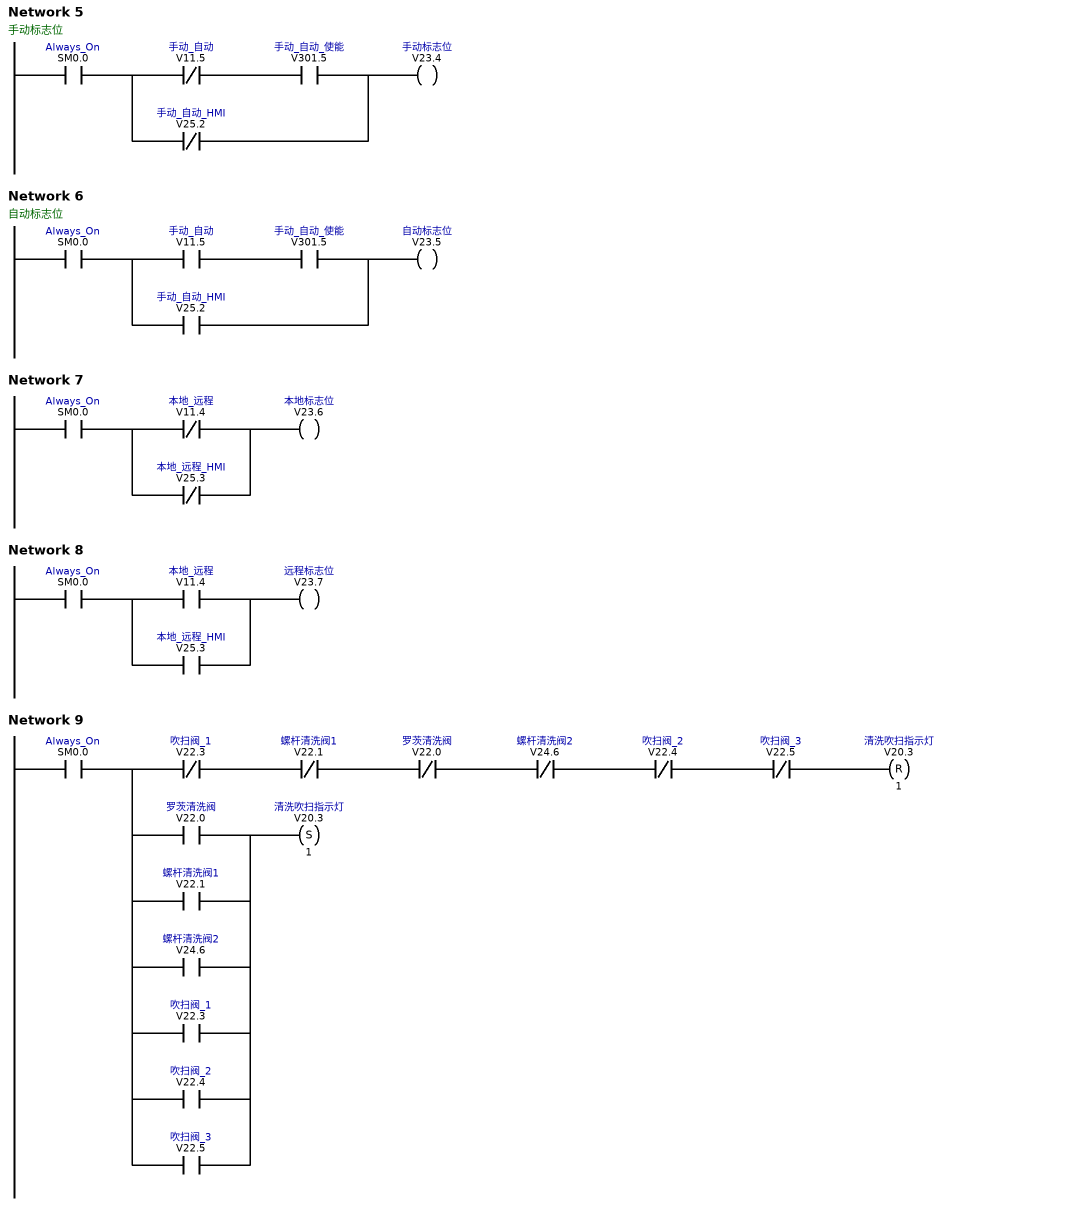
[picture p24: SBR11 networks 5-9]
Network 5
// 手动标志位
LD     Always_On:SM0.0
LDN    手动_自动:V11.5
A      手动_自动_使能:V301.5
ON     手动_自动_HMI:V25.2
ALD
=      手动标志位:V23.4
Network 6
// 自动标志位
LD     Always_On:SM0.0
LD     手动_自动:V11.5
A      手动_自动_使能:V301.5
O      手动_自动_HMI:V25.2
ALD
=      自动标志位:V23.5
Network 7
LD     Always_On:SM0.0
LDN    本地_远程:V11.4
ON     本地_远程_HMI:V25.3
ALD
=      本地标志位:V23.6
Network 8
LD     Always_On:SM0.0
LD     本地_远程:V11.4
O      本地_远程_HMI:V25.3
ALD
=      远程标志位:V23.7
Network 9
LD     Always_On:SM0.0
LPS
AN     吹扫阀_1:V22.3
AN     螺杆清洗阀1:V22.1
AN     罗茨清洗阀:V22.0
AN     螺杆清洗阀2:V24.6
AN     吹扫阀_2:V22.4
AN     吹扫阀_3:V22.5
R      清洗吹扫指示灯:V20.3, 1
LPP
LD     罗茨清洗阀:V22.0
O      螺杆清洗阀1:V22.1
O      螺杆清洗阀2:V24.6
O      吹扫阀_1:V22.3
O      吹扫阀_2:V22.4
O      吹扫阀_3:V22.5
ALD
S      清洗吹扫指示灯:V20.3, 1
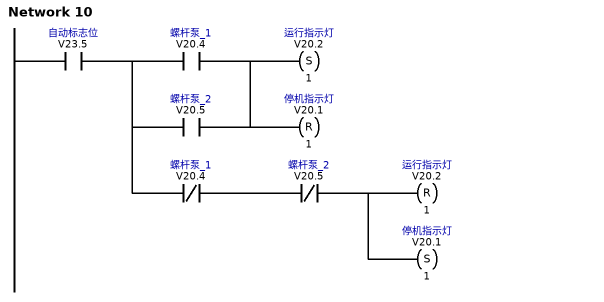
Network 10
LD     自动标志位:V23.5
LPS
LD     螺杆泵_1:V20.4
O      螺杆泵_2:V20.5
ALD
S      运行指示灯:V20.2, 1
R      停机指示灯:V20.1, 1
LPP
AN     螺杆泵_1:V20.4
AN     螺杆泵_2:V20.5
R      运行指示灯:V20.2, 1
S      停机指示灯:V20.1, 1
END_SUBROUTINE_BLOCK

SUBROUTINE_BLOCK C_真空度转化:SBR12
TITLE=子程序注释
VAR_INPUT
输入真空:REAL;	// LD0 
END_VAR
VAR_OUTPUT
输出负压:REAL;	// LD4 
END_VAR
VAR
中间变量:REAL;	// LD8 
END_VAR
BEGIN
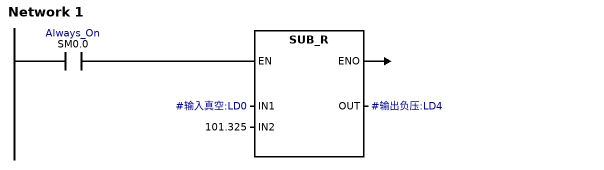
Network 1
LD     Always_On:SM0.0
MOVR   #输入真空:LD0, #输出负压:LD4
-R     101.325, #输出负压:LD4
END_SUBROUTINE_BLOCK

SUBROUTINE_BLOCK C_1套运行时间:SBR13
TITLE=子程序注释
VAR_INPUT
电机:BOOL;	// L0.0 
清零:BOOL;	// L0.1 
秒脉冲:BOOL;	// L0.2 
END_VAR
VAR_IN_OUT
秒:INT;	// LW1 
分:INT;	// LW3 
时:INT;	// LW5 
END_VAR
BEGIN
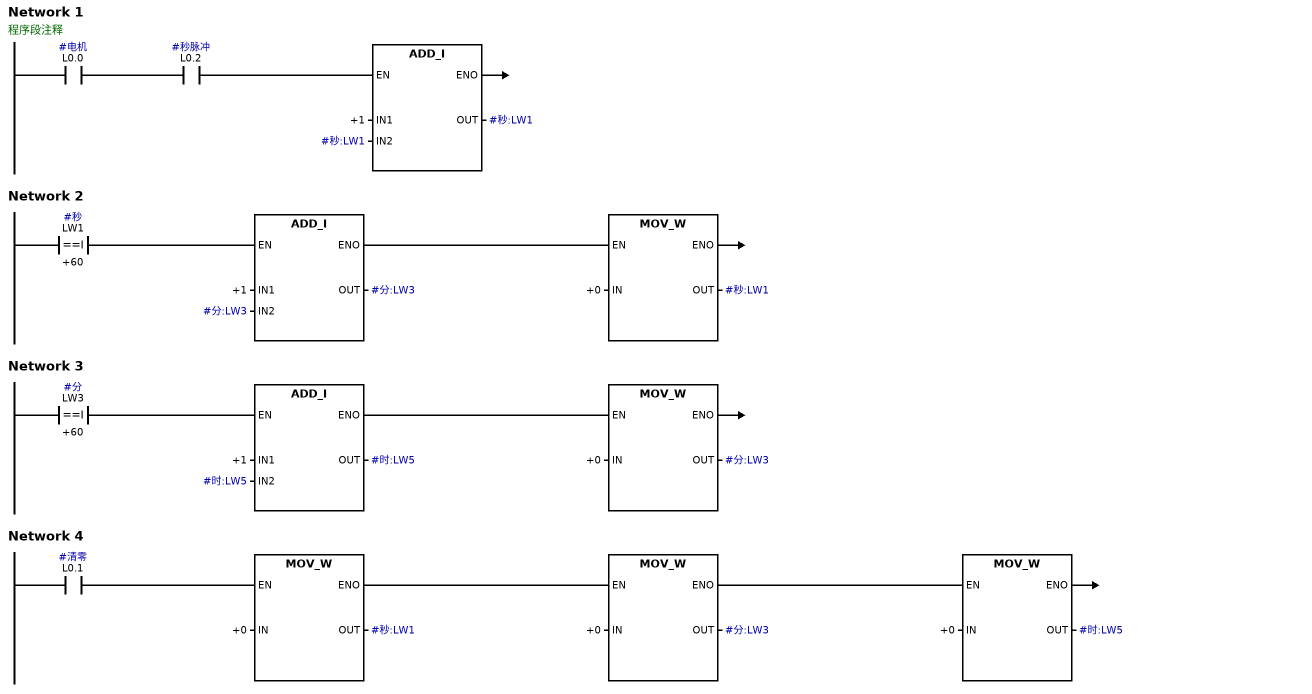
Network 1
// 程序段注释
LD     #电机:L0.0
A      #秒脉冲:L0.2
+I     +1, #秒:LW1
Network 2
LDW=   #秒:LW1, +60
+I     +1, #分:LW3
AENO
MOVW   +0, #秒:LW1
Network 3
LDW=   #分:LW3, +60
+I     +1, #时:LW5
AENO
MOVW   +0, #分:LW3
Network 4
LD     #清零:L0.1
MOVW   +0, #秒:LW1
AENO
MOVW   +0, #分:LW3
AENO
MOVW   +0, #时:LW5
END_SUBROUTINE_BLOCK

SUBROUTINE_BLOCK C_2套运行时间:SBR15
TITLE=子程序注释
VAR_INPUT
清零:BOOL;	// L0.0 
秒脉冲:BOOL;	// L0.1 
电机2:BOOL;	// L0.2 
电机1:BOOL;	// L0.3 
END_VAR
VAR_IN_OUT
秒1:INT;	// LW1 
分1:INT;	// LW3 
时1:INT;	// LW5 
秒2:INT;	// LW7 
分2:INT;	// LW9 
时2:INT;	// LW11 
END_VAR
BEGIN
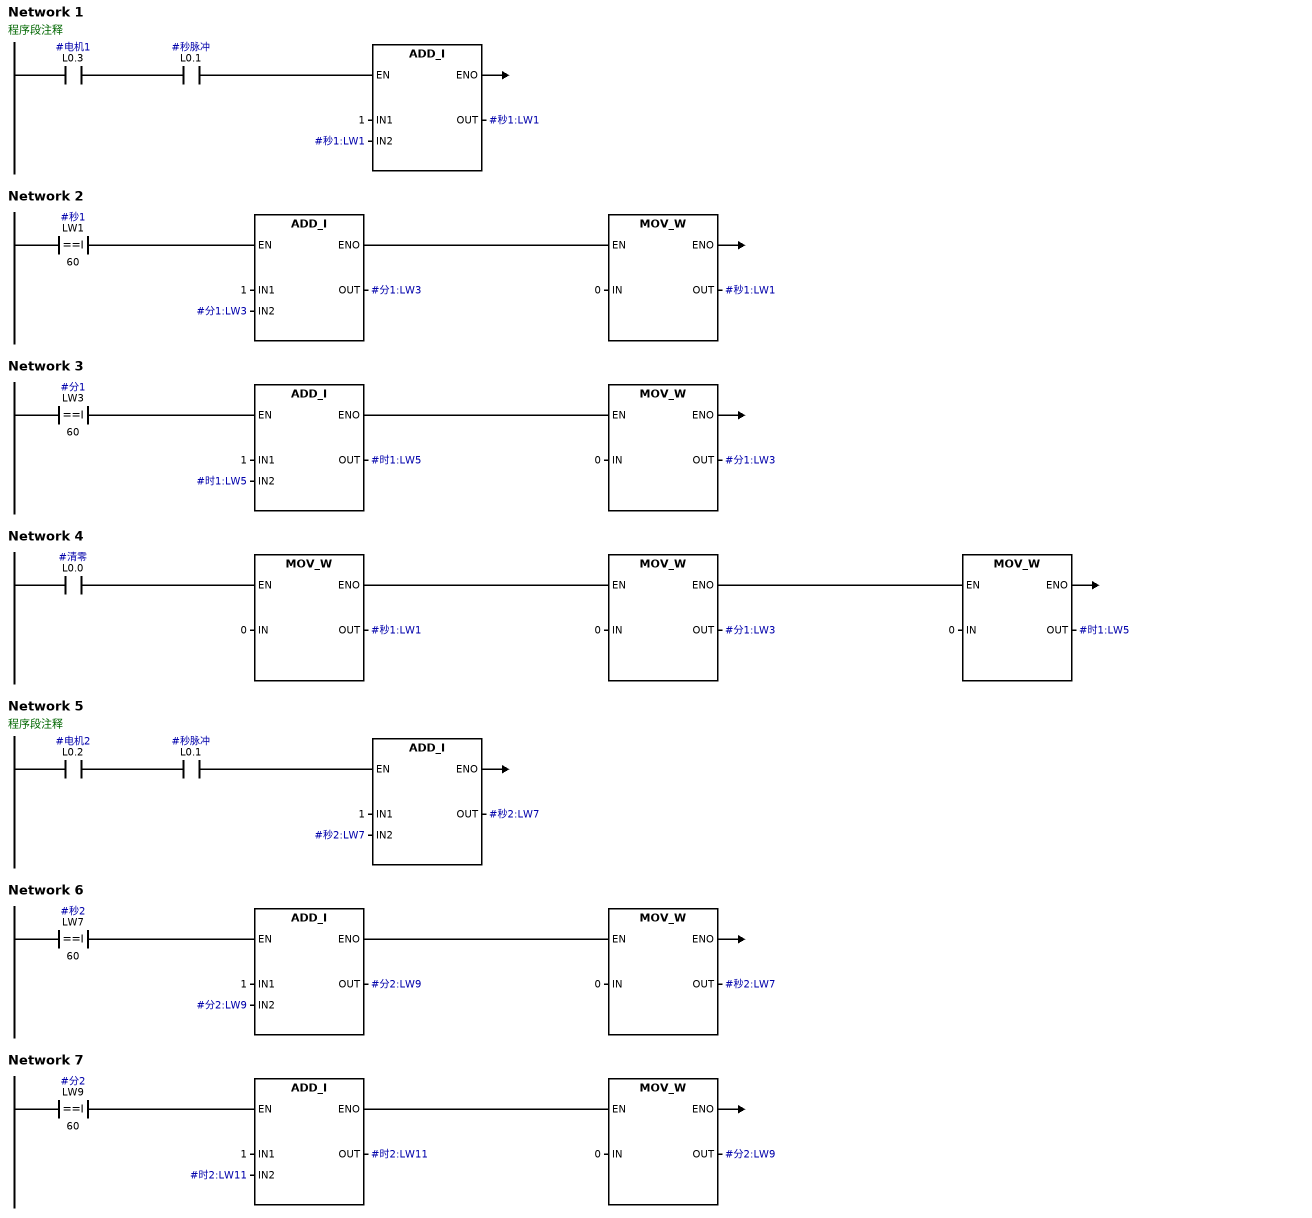
Network 1
// 程序段注释
LD     #电机1:L0.3
A      #秒脉冲:L0.1
+I     1, #秒1:LW1
Network 2
LDW=   #秒1:LW1, 60
+I     1, #分1:LW3
AENO
MOVW   0, #秒1:LW1
Network 3
LDW=   #分1:LW3, 60
+I     1, #时1:LW5
AENO
MOVW   0, #分1:LW3
Network 4
LD     #清零:L0.0
MOVW   0, #秒1:LW1
AENO
MOVW   0, #分1:LW3
AENO
MOVW   0, #时1:LW5
Network 5
// 程序段注释
LD     #电机2:L0.2
A      #秒脉冲:L0.1
+I     1, #秒2:LW7
Network 6
LDW=   #秒2:LW7, 60
+I     1, #分2:LW9
AENO
MOVW   0, #秒2:LW7
Network 7
LDW=   #分2:LW9, 60
+I     1, #时2:LW11
AENO
MOVW   0, #分2:LW9
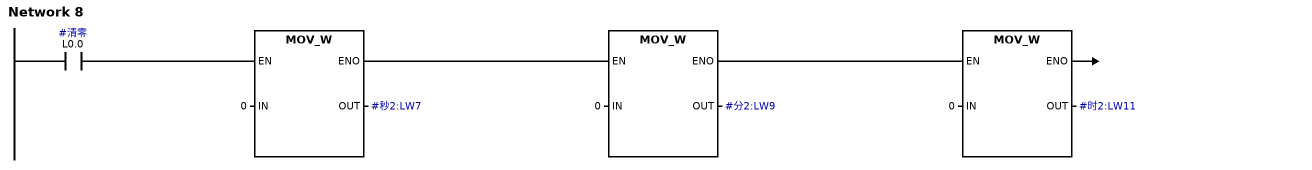
Network 8
LD     #清零:L0.0
MOVW   0, #秒2:LW7
AENO
MOVW   0, #分2:LW9
AENO
MOVW   0, #时2:LW11
END_SUBROUTINE_BLOCK

SUBROUTINE_BLOCK C_变频_单螺杆机组A:SBR17
TITLE=子程序注释
BEGIN
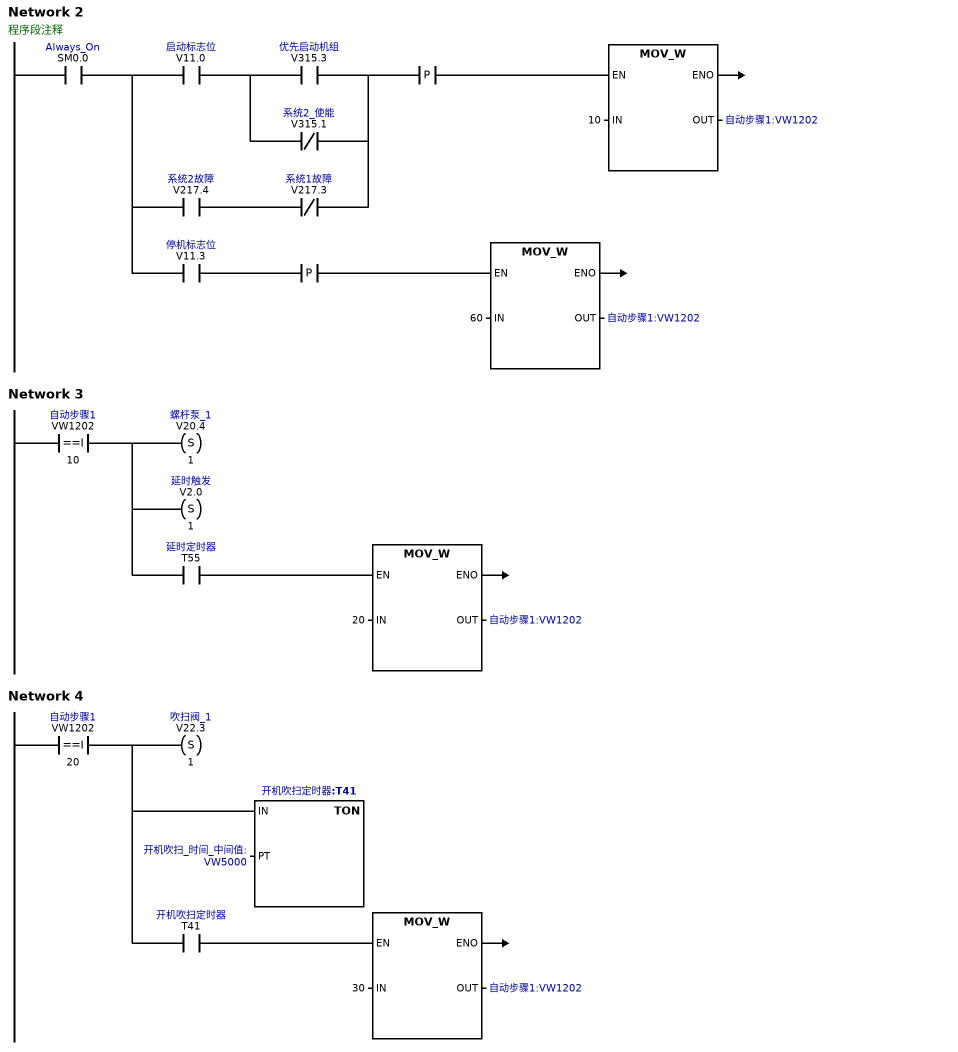
Network 2
// 程序段注释
LD     Always_On:SM0.0
LPS
LD     启动标志位:V11.0
LD     优先启动机组:V315.3
ON     系统2_使能:V315.1
ALD
LD     系统2故障:V217.4
AN     系统1故障:V217.3
OLD
ALD
EU
MOVW   10, 自动步骤1:VW1202
LPP
A      停机标志位:V11.3
EU
MOVW   60, 自动步骤1:VW1202
Network 3
LDW=   自动步骤1:VW1202, 10
S      螺杆泵_1:V20.4, 1
S      延时触发:V2.0, 1
A      延时定时器:T55
MOVW   20, 自动步骤1:VW1202
Network 4
LDW=   自动步骤1:VW1202, 20
S      吹扫阀_1:V22.3, 1
TON    开机吹扫定时器:T41, 开机吹扫_时间_中间值:VW5000
A      开机吹扫定时器:T41
MOVW   30, 自动步骤1:VW1202
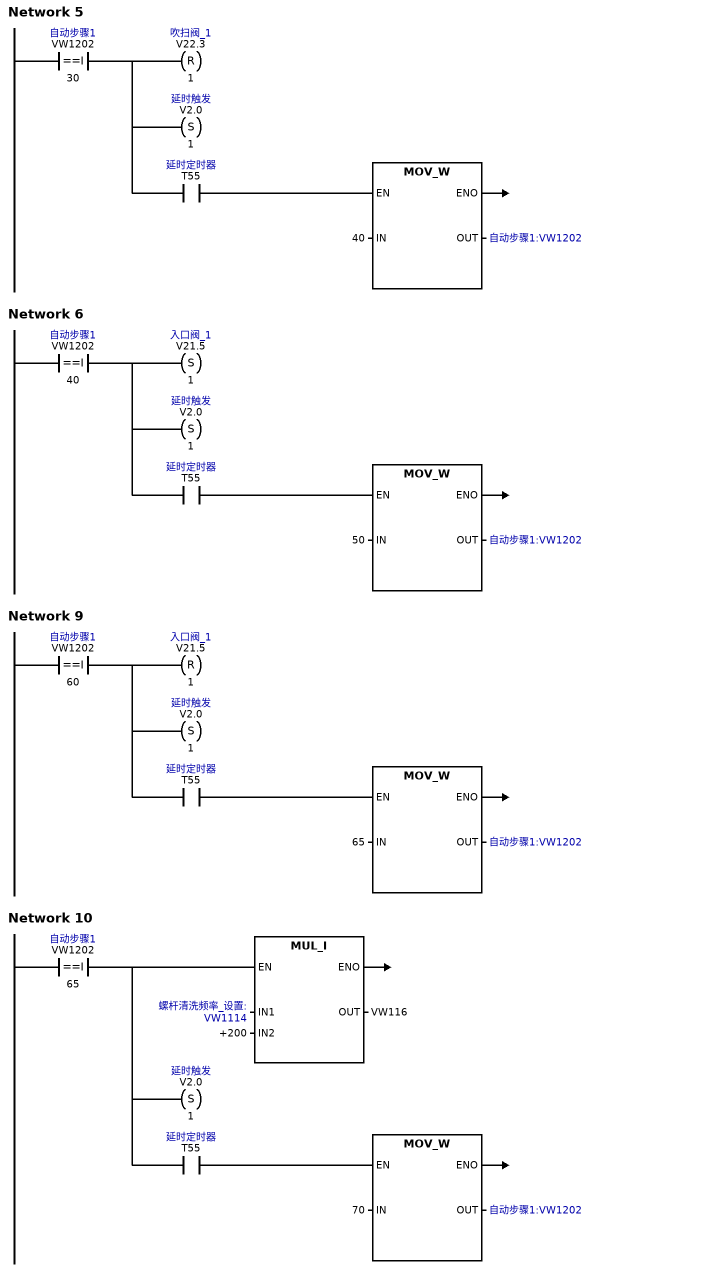
Network 5
LDW=   自动步骤1:VW1202, 30
R      吹扫阀_1:V22.3, 1
S      延时触发:V2.0, 1
A      延时定时器:T55
MOVW   40, 自动步骤1:VW1202
Network 6
LDW=   自动步骤1:VW1202, 40
S      入口阀_1:V21.5, 1
S      延时触发:V2.0, 1
A      延时定时器:T55
MOVW   50, 自动步骤1:VW1202
Network 9
LDW=   自动步骤1:VW1202, 60
R      入口阀_1:V21.5, 1
S      延时触发:V2.0, 1
A      延时定时器:T55
MOVW   65, 自动步骤1:VW1202
Network 10
LDW=   自动步骤1:VW1202, 65
MOVW   螺杆清洗频率_设置:VW1114, VW116
*I     +200, VW116
S      延时触发:V2.0, 1
A      延时定时器:T55
MOVW   70, 自动步骤1:VW1202
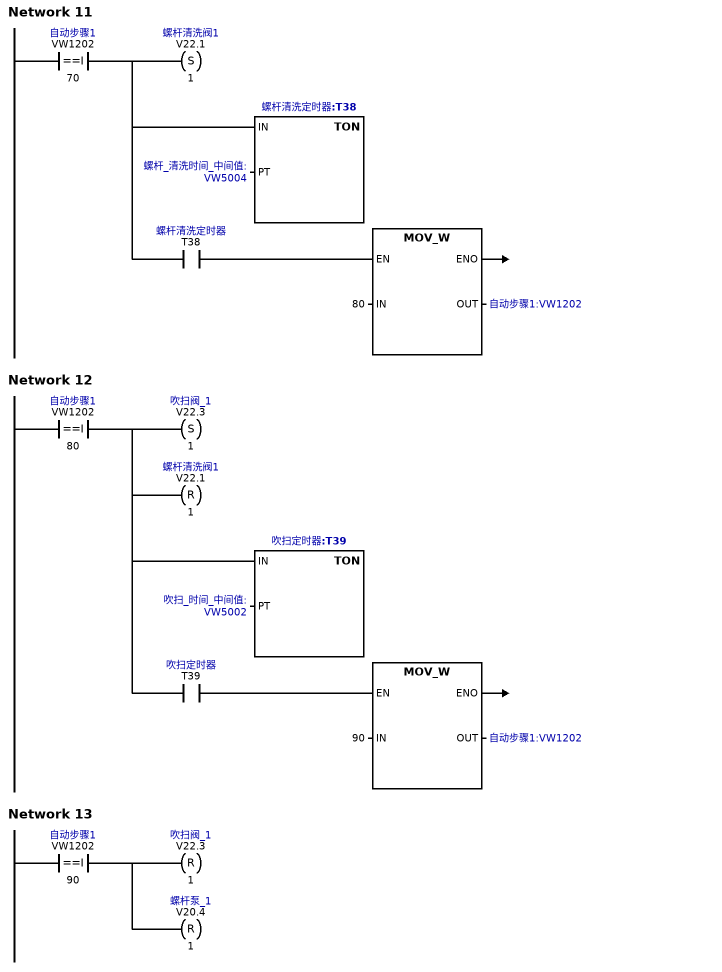
Network 11
LDW=   自动步骤1:VW1202, 70
S      螺杆清洗阀1:V22.1, 1
TON    螺杆清洗定时器:T38, 螺杆_清洗时间_中间值:VW5004
A      螺杆清洗定时器:T38
MOVW   80, 自动步骤1:VW1202
Network 12
LDW=   自动步骤1:VW1202, 80
S      吹扫阀_1:V22.3, 1
R      螺杆清洗阀1:V22.1, 1
TON    吹扫定时器:T39, 吹扫_时间_中间值:VW5002
A      吹扫定时器:T39
MOVW   90, 自动步骤1:VW1202
Network 13
LDW=   自动步骤1:VW1202, 90
R      吹扫阀_1:V22.3, 1
R      螺杆泵_1:V20.4, 1
END_SUBROUTINE_BLOCK

// SBR18: protected block, not included

// SBR19: protected block, not included

SUBROUTINE_BLOCK C_变频_单螺杆机组B:SBR20
TITLE=
BEGIN
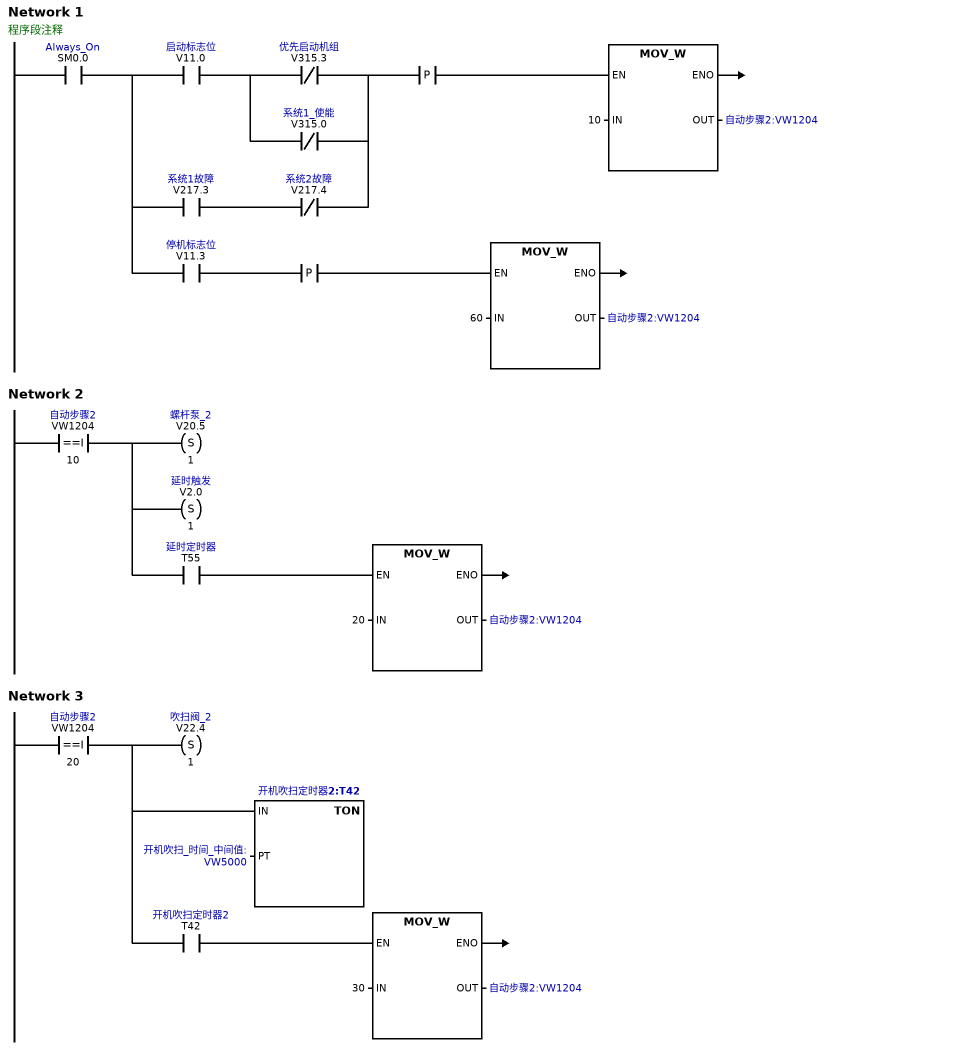
Network 1
// 程序段注释
LD     Always_On:SM0.0
LPS
LD     启动标志位:V11.0
LDN    优先启动机组:V315.3
ON     系统1_使能:V315.0
ALD
LD     系统1故障:V217.3
AN     系统2故障:V217.4
OLD
ALD
EU
MOVW   10, 自动步骤2:VW1204
LPP
A      停机标志位:V11.3
EU
MOVW   60, 自动步骤2:VW1204
Network 2
LDW=   自动步骤2:VW1204, 10
S      螺杆泵_2:V20.5, 1
S      延时触发:V2.0, 1
A      延时定时器:T55
MOVW   20, 自动步骤2:VW1204
Network 3
LDW=   自动步骤2:VW1204, 20
S      吹扫阀_2:V22.4, 1
TON    开机吹扫定时器2:T42, 开机吹扫_时间_中间值:VW5000
A      开机吹扫定时器2:T42
MOVW   30, 自动步骤2:VW1204
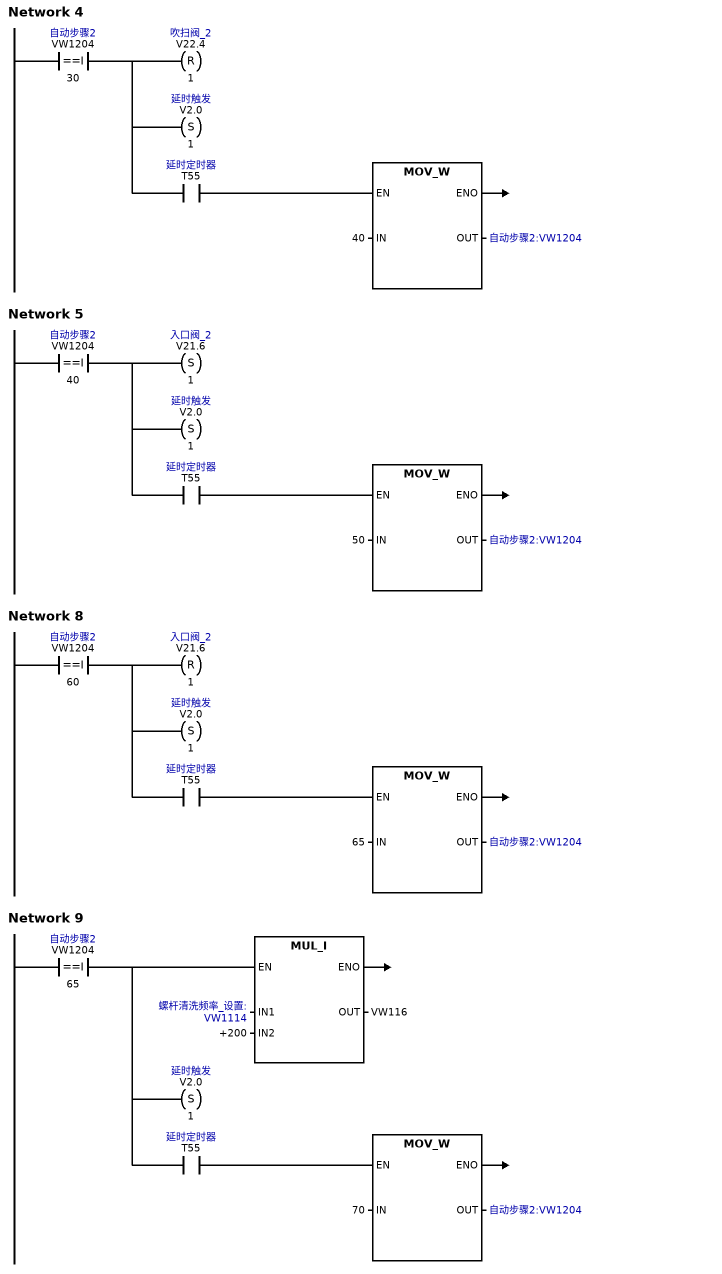
Network 4
LDW=   自动步骤2:VW1204, 30
R      吹扫阀_2:V22.4, 1
S      延时触发:V2.0, 1
A      延时定时器:T55
MOVW   40, 自动步骤2:VW1204
Network 5
LDW=   自动步骤2:VW1204, 40
S      入口阀_2:V21.6, 1
S      延时触发:V2.0, 1
A      延时定时器:T55
MOVW   50, 自动步骤2:VW1204
Network 8
LDW=   自动步骤2:VW1204, 60
R      入口阀_2:V21.6, 1
S      延时触发:V2.0, 1
A      延时定时器:T55
MOVW   65, 自动步骤2:VW1204
Network 9
LDW=   自动步骤2:VW1204, 65
MOVW   螺杆清洗频率_设置:VW1114, VW116
*I     +200, VW116
S      延时触发:V2.0, 1
A      延时定时器:T55
MOVW   70, 自动步骤2:VW1204
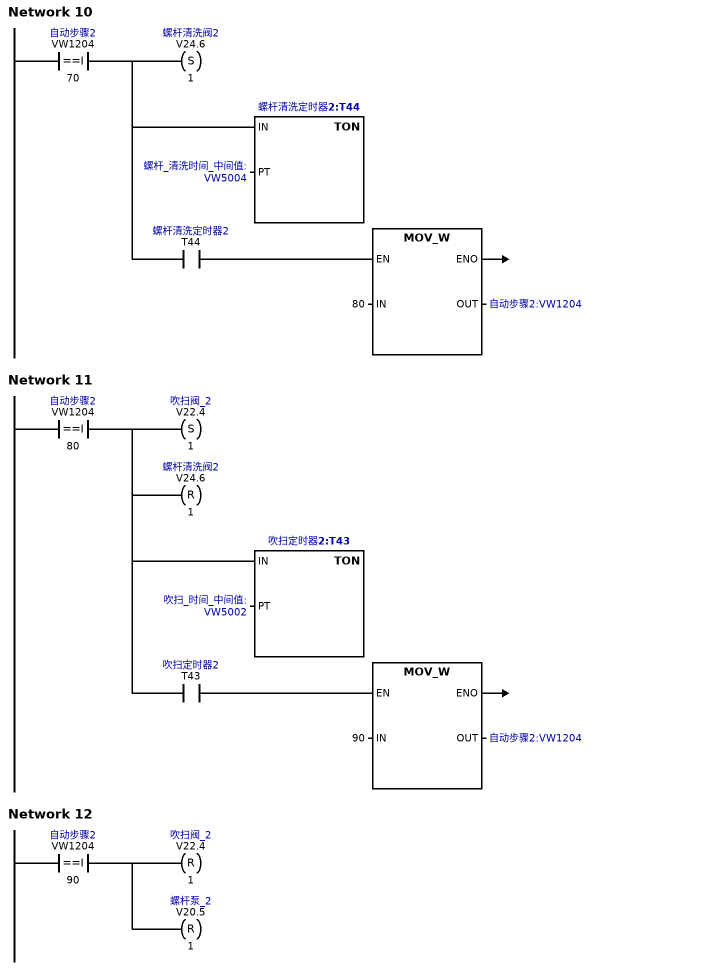
Network 10
LDW=   自动步骤2:VW1204, 70
S      螺杆清洗阀2:V24.6, 1
TON    螺杆清洗定时器2:T44, 螺杆_清洗时间_中间值:VW5004
A      螺杆清洗定时器2:T44
MOVW   80, 自动步骤2:VW1204
Network 11
LDW=   自动步骤2:VW1204, 80
S      吹扫阀_2:V22.4, 1
R      螺杆清洗阀2:V24.6, 1
TON    吹扫定时器2:T43, 吹扫_时间_中间值:VW5002
A      吹扫定时器2:T43
MOVW   90, 自动步骤2:VW1204
Network 12
LDW=   自动步骤2:VW1204, 90
R      吹扫阀_2:V22.4, 1
R      螺杆泵_2:V20.5, 1
END_SUBROUTINE_BLOCK

SUBROUTINE_BLOCK A_定时器_时间转换:SBR21
TITLE=子程序注释
BEGIN
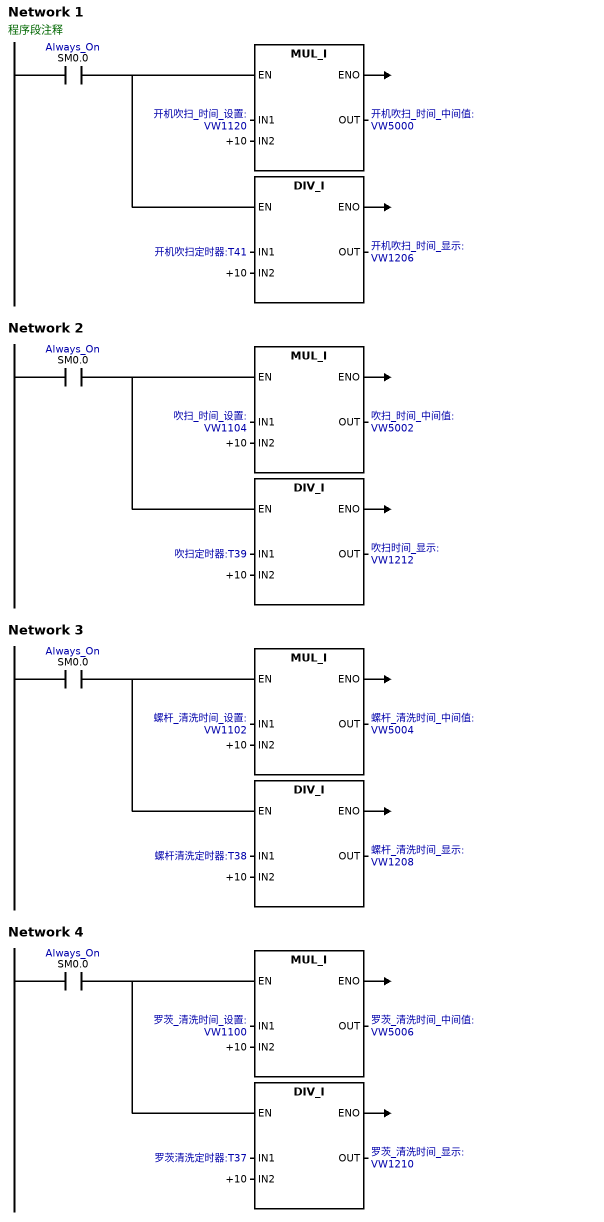
Network 1
// 程序段注释
LD     Always_On:SM0.0
MOVW   开机吹扫_时间_设置:VW1120, 开机吹扫_时间_中间值:VW5000
*I     +10, 开机吹扫_时间_中间值:VW5000
MOVW   开机吹扫定时器:T41, 开机吹扫_时间_显示:VW1206
/I     +10, 开机吹扫_时间_显示:VW1206
Network 2
LD     Always_On:SM0.0
MOVW   吹扫_时间_设置:VW1104, 吹扫_时间_中间值:VW5002
*I     +10, 吹扫_时间_中间值:VW5002
MOVW   吹扫定时器:T39, 吹扫时间_显示:VW1212
/I     +10, 吹扫时间_显示:VW1212
Network 3
LD     Always_On:SM0.0
MOVW   螺杆_清洗时间_设置:VW1102, 螺杆_清洗时间_中间值:VW5004
*I     +10, 螺杆_清洗时间_中间值:VW5004
MOVW   螺杆清洗定时器:T38, 螺杆_清洗时间_显示:VW1208
/I     +10, 螺杆_清洗时间_显示:VW1208
Network 4
LD     Always_On:SM0.0
MOVW   罗茨_清洗时间_设置:VW1100, 罗茨_清洗时间_中间值:VW5006
*I     +10, 罗茨_清洗时间_中间值:VW5006
MOVW   罗茨清洗定时器:T37, 罗茨_清洗时间_显示:VW1210
/I     +10, 罗茨_清洗时间_显示:VW1210
END_SUBROUTINE_BLOCK

SUBROUTINE_BLOCK B_PID调节:SBR22
TITLE=子程序注释
BEGIN
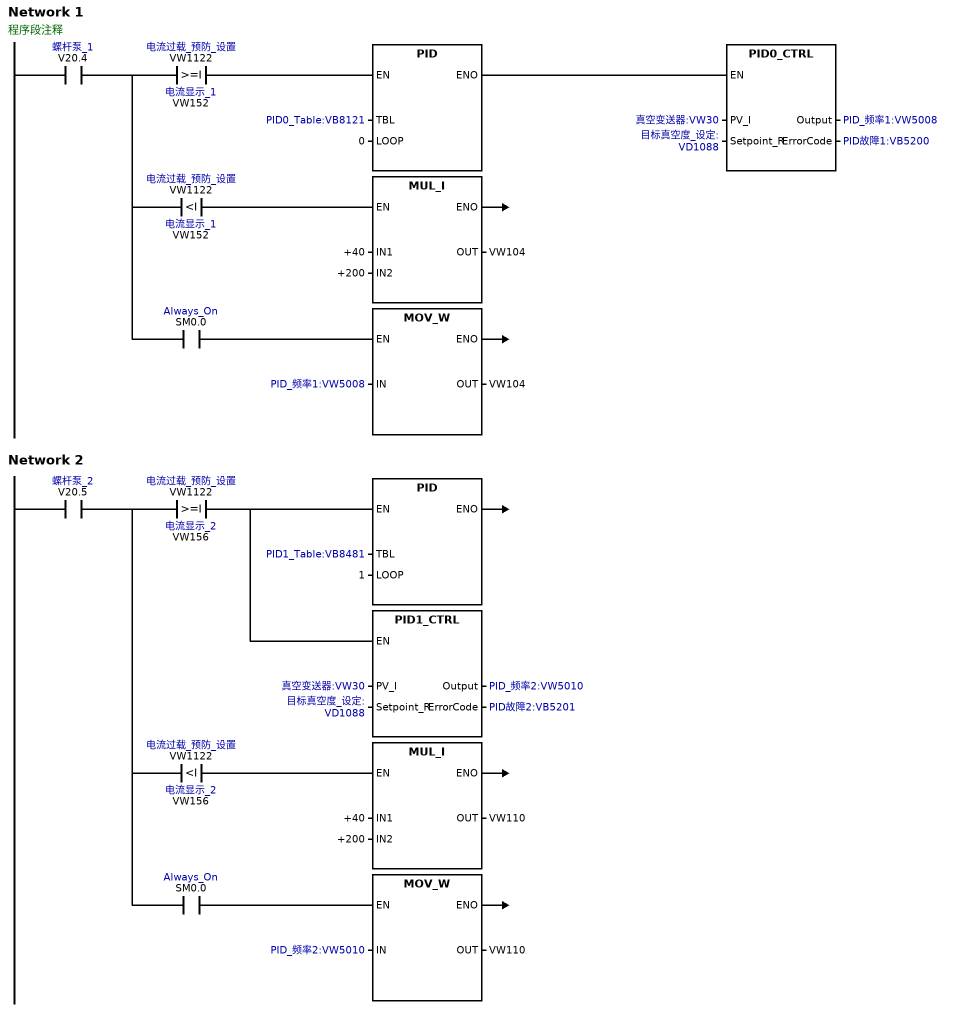
Network 1
// 程序段注释
LD     螺杆泵_1:V20.4
LPS
AW>=   电流过载_预防_设置:VW1122, 电流显示_1:VW152
PID    PID0_Table:VB8121, 0
AENO
CALL   PID0_CTRL:SBR18, 真空变送器:VW30, 目标真空度_设定:VD1088, PID_频率1:VW5008, PID故障1:VB5200
LRD
AW<    电流过载_预防_设置:VW1122, 电流显示_1:VW152
MOVW   +40, VW104
*I     +200, VW104
LPP
A      Always_On:SM0.0
MOVW   PID_频率1:VW5008, VW104
Network 2
LD     螺杆泵_2:V20.5
LPS
AW>=   电流过载_预防_设置:VW1122, 电流显示_2:VW156
PID    PID1_Table:VB8481, 1
CALL   PID1_CTRL:SBR19, 真空变送器:VW30, 目标真空度_设定:VD1088, PID_频率2:VW5010, PID故障2:VB5201
LPP
LPS
AW<    电流过载_预防_设置:VW1122, 电流显示_2:VW156
MOVW   +40, VW110
*I     +200, VW110
LPP
A      Always_On:SM0.0
MOVW   PID_频率2:VW5010, VW110
END_SUBROUTINE_BLOCK

DATA_BLOCK_TAB 页面_1
BEGIN
//参数设置
//报警保护参数
//低于该液位值关闭排污阀
//变送器基本配置
         罗茨_温度报警_设置, 45.0
         罗茨_温度停机_设置, 55.0
         电流_保护_设置, 43.7
         电流过载_预防_设置, 44
         螺杆_温度停机_设置, 55.0
         电流_恢复_设置, 15.0
         液位_保护_设置, 300.0
         液位_恢复_设置, 200.0
         液位_变送器上限_设置, 350.0
         螺杆温度_变送器上限_设, 100.0
         电流_变送器上限_设置, 50.0
         罗茨1温度_变送器上限_设, 100.0
         罗茨2温度_变送器上限_设, 100.0
         罗茨1启动真空设定, 8.0
         罗茨1停机真空设定, 10.0
         罗茨2启动真空设定, 4.0
         罗茨2停机真空设定, 7.0
         真空_变送器上限_设定, 130.0
         氮气_变送器上限_设定, 4.0
         氮气_低压急停_设定, 0.3
         氮气_低压报警_设定, 0.6
         目标真空度_设定, 0.0
//清洗吹扫参数设置
         螺杆_清洗时间_设置, 600     //毫秒
         吹扫_时间_设置, 600
         开机吹扫_时间_设置, 300
//毫秒
//毫秒
         液位_过高报警_设置, 200.0
         螺杆_温度报警_设置, 45.0
         螺杆手动频率_设置, 50
         罗茨1手动频率_设置, 50
         罗茨2手动频率_设置, 50
         螺杆2手动频率_设置, 50
         螺杆清洗频率_设置, 30
END_DATA_BLOCK_TAB
